// TIA Portal project "FactoryIO_Template_S7-1200_V16_V16" (V16)
// Vorlageprojekt für das Buch mit Zielsystem S7-1200

(* hardware
DEVICE "S7-1200-Station_1"  S7-1200 Station
   slot 0: "Baugruppenträger_0"  Rack  V1.0
   slot 1: "PLC_1"  CPU 1211C DC/DC/DC  6ES7 211-1AE40-0XB0  V4.1
*)

// ===== PLC "PLC_1"  CPU 1211C DC/DC/DC =====

VAR_GLOBAL   // PLC tag table "Standard-Variablentabelle"
   "Tag_1" AT %Q0.1 : Bool;
   "Tag_2" AT %E0.0 : Bool;
   "Tag_3" AT %E0.1 : Bool;
   "start" AT %I10.0 : Bool;
   "Tag_5" AT %Q0.0 : Bool;
   "stop" AT %I0.1 : Bool;
   "Tag_7" AT %Q0.1 : Bool;
   "Tag_8" AT %M0.1 : Bool;
   "KK" AT %I0.3 : Bool;
   "Tag_10" AT %Q0.3 : Bool;
   "Tag_4" AT %I0.4 : Bool;
   "Tag_6" AT %Q0.4 : Bool;
   "Tag_9" AT %Q0.5 : Bool;
   "Tag_11" AT %I0.3 : Bool;
   "Tag_12" AT %Q10.7 : Bool;
   "Tag_13" AT %Q10.7 : Bool;
   "Tag_14" AT %Q0.7 : Bool;
   "Tag_15" AT %Q1.0 : Bool;
   "Tag_16" AT %Q1.1 : Bool;
   "Tag_17" AT %Q1.2 : Bool;
   "Tag_18" AT %I0.5 : Bool;
   "Tag_19" AT %Q1.3 : Bool;
   "Tag_20" AT %Q1.4 : Bool;
   "Tag_21" AT %Q0.6 : Bool;
   "START(1)" AT %I0.0 : Bool;
   "Tag_22" AT %I0.1 : Bool;
   "Tag_23" AT %M0.1 : Bool;
   "Tag_24" AT %Q0.2 : Bool;
   "Tag_25" AT %M0.0 : Bool;
END_VAR

FUNCTION "MHJ-PLC-Lab-Function-S71200" : Void   // FC9000, SCL
{ S7_Optimized_Access := 'TRUE' }
VERSION : 0.1
   VAR_TEMP
      rdTimeReturn : Int;
      outputTime : DTL;
      SyncVal : Byte;
      forVal : Int;
      forVal_2 : Int;
      Value : Byte;
   END_VAR
   VAR CONSTANT
      CompVal : Byte := 16#34;
      Value_01 : Byte := 16#11;
      Value_01_DW : DWord := 16#A165_D992;
      Value_02_DW : DWord := 16#58BE_4401;
   END_VAR
BEGIN

   #Value:=PEEK(area := 16#82,
        dbNumber := 0,
        byteOffset := 511);
   #Value := #Value + 1;

   POKE(area := 16#82,
        dbNumber := 0,
        byteOffset := 511,
        value := #Value);

   POKE(area:=16#81,
        dbNumber:=0,
        byteOffset:=1016,
        value:=#Value_01_DW);
   POKE(area := 16#81,
        dbNumber := 0,
        byteOffset := 1020,
        value := #Value_02_DW);

   POKE(area := 16#81,
        dbNumber := 0,
        byteOffset := 511,
        value := B#16#00);

   FOR #forVal := 0 TO 120 DO
       FOR #forVal_2:=0 TO 10 DO
           #rdTimeReturn:=RD_SYS_T(#outputTime);
           #rdTimeReturn := WR_SYS_T(#outputTime);
           #rdTimeReturn := RD_SYS_T(#outputTime);
           #rdTimeReturn := WR_SYS_T(#outputTime);
       END_FOR;
       #SyncVal:= PEEK(area := 16#81,
                      dbNumber := 0,
                      byteOffset := 511);
       IF #SyncVal = #CompVal THEN
          GOTO M_1;
       END_IF;
   END_FOR;
   RETURN;

   M_1:
   POKE(area := 16#81,
        dbNumber := 0,
        byteOffset := 511,
        value := B#16#0);
END_FUNCTION

ORGANIZATION_BLOCK "Main"   // OB1, LAD, ProgramCycle
TITLE = "Main Program Sweep (Cycle)"
{ S7_Optimized_Access := 'TRUE' }
VERSION : 0.1
   VAR_INPUT
      Initial_Call : Bool;   // Initial call of this OB
      Remanence : Bool;   // =True, if remanent data are available
   END_VAR
BEGIN

REGION Network 1: Konnektierungsbaustein für PLC-Lab
   // Im Netzwerk 1 wird der Konnektierungsbaustein für PLC-Lab aufgerufen.
   // Dieser Aufruf darf nicht entfernt werden!
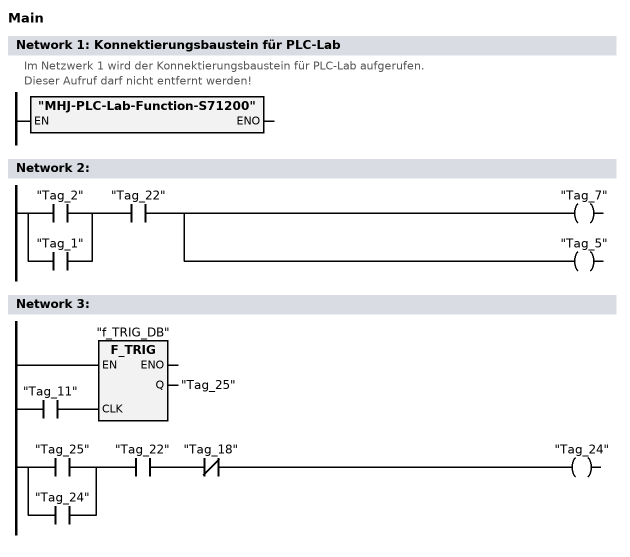
   RUNG wire#powerrail
      "MHJ-PLC-Lab-Function-S71200"()
   END_RUNG
   // the same network as SCL:
   "MHJ-PLC-Lab-Function-S71200"();
END_REGION

REGION Network 2
   RUNG wire#powerrail
      Contact( "Tag_2" )
      wire#w1
      Contact( "Tag_22" )
      wire#w2
      Coil( "Tag_7" )
   END_RUNG
   RUNG wire#powerrail
      Contact( "Tag_1" )
   END_RUNG wire#w1
   RUNG wire#w2
      Coil( "Tag_5" )
   END_RUNG
   // the same network as SCL:
   "Tag_7" := ("Tag_2" OR "Tag_1") AND "Tag_22";
   "Tag_5" := "Tag_7";
END_REGION

REGION Network 3
   "f_TRIG_DB"(CLK := "Tag_11", Q => "Tag_25");   // F_TRIG
   "Tag_24" := ("Tag_25" OR "Tag_24") AND "Tag_22" AND NOT "Tag_18";
END_REGION
END_ORGANIZATION_BLOCK